// TIA Portal V20 export
TYPE "IO_Device_Test_Parameters"
   STRUCT
      Reset_PLC_Functional_Test_1 : Bool;
      Reset_PLC_Functional_Test_3 : Bool;
      Reset_PLC_Functional_Test_5 : Bool;
      Reset_PLC_Functional_Test_7 : Bool;
      Reset_PLC_Functional_Test_9 : Bool;
      Reset_PLC_Functional_Test_11 : Bool;
      Reset_PLC_Functional_Test_13 : Bool;
      Reset_PLC_Functional_Test_15 : Bool;
      Reset_PLC_Functional_Test_17 : Bool;
      Reset_PLC_Functional_Test_19 : Bool;
      Reset_PLC_Functional_Test_21 : Bool;
      Reset_PLC_Functional_Test_23 : Bool;
      Reset_PLC_Functional_Test_25 : Bool;
      Reset_PLC_Functional_Test_27 : Bool;
      Reset_PLC_Functional_Test_29 : Bool;
      Status : Bool;
      Voltage_Read : UInt;
      Min_Electrical_Current : UInt;
      Max_Electrical_Current : UInt;
      Time_End_Electrical_Current_Test : Time;
      Time_Start_Visual_Test : Time;
   END_STRUCT;
END_TYPE
